(* PLC project poST.project, poSTIDE *)
(* stored: creationDateTime 2021-08-31T00:00:00.000000 *)

FUNCTION EXPT : ANY_REAL
  VAR_INPUT
    in1 : ANY_REAL;
    in2 : ANY_REAL;
  END_VAR

END_FUNCTION
